(* PLC project batch, Dassault Systèmes ControlBuild 2024x Refresh1 *)
(* stored: creationDateTime 2024-03-18T16:40:20-01:00 *)

FUNCTION_BLOCK acknowledgepb
  VAR_IN_OUT
    action : BOOL := false;
    timeCounter : REAL := 0.0;
    pulseDuration : REAL := 0.0;
    PBLogic : BOOL := false;
  END_VAR
  VAR_OUTPUT
    PB : BOOL := false;
  END_VAR


ACTION C_source_code:

END_ACTION
END_FUNCTION_BLOCK

FUNCTION_BLOCK bpcloture
  VAR_IN_OUT
    action : BOOL := false;
    timeCounter : REAL := 0.0;
    pulseDuration : REAL := 0.0;
    PBLogic : BOOL := false;
  END_VAR
  VAR_OUTPUT
    PB : BOOL := false;
  END_VAR


ACTION C_source_code:

END_ACTION
END_FUNCTION_BLOCK

FUNCTION_BLOCK emergencystop
  VAR_IN_OUT
    action : BOOL := false;
    PBLogic : BOOL := false;
  END_VAR
  VAR_OUTPUT
    pb : BOOL := false;
  END_VAR


ACTION C_source_code:

END_ACTION
END_FUNCTION_BLOCK

FUNCTION_BLOCK endcyclepb
  VAR_IN_OUT
    action : BOOL := false;
    timeCounter : REAL := 0.0;
    pulseDuration : REAL := 0.0;
    PBLogic : BOOL := false;
  END_VAR
  VAR_OUTPUT
    PB : BOOL := false;
  END_VAR


ACTION C_source_code:

END_ACTION
END_FUNCTION_BLOCK

FUNCTION_BLOCK modeswitch
  VAR_IN_OUT
    leftPosition : BOOL := false;
    rightPosition : BOOL := false;
  END_VAR
  VAR_OUTPUT
    leftVariable : BOOL := false;
    rightVariable : BOOL := false;
  END_VAR


ACTION C_source_code:

END_ACTION
END_FUNCTION_BLOCK

FUNCTION_BLOCK powerup
  VAR_IN_OUT
    action : BOOL := false;
    timeCounter : REAL := 0.0;
    pulseDuration : REAL := 0.0;
    PBLogic : BOOL := false;
  END_VAR
  VAR_OUTPUT
    PB : BOOL := false;
  END_VAR


ACTION C_source_code:

END_ACTION
END_FUNCTION_BLOCK

FUNCTION_BLOCK startcyclepb
  VAR_IN_OUT
    action : BOOL := false;
    timeCounter : REAL := 0.0;
    pulseDuration : REAL := 0.0;
    PBLogic : BOOL := false;
  END_VAR
  VAR_OUTPUT
    PB : BOOL := false;
  END_VAR


ACTION C_source_code:

END_ACTION
END_FUNCTION_BLOCK

PROGRAM generalpanel
  VAR_OUTPUT
    acknowledgePB : BOOL := false;
    powerUp : BOOL := false;
    emergencyStop : BOOL := false;
    manualSwitch : BOOL := false;
    autoSwitch : BOOL := false;
    startCyclePB : BOOL := false;
    endCyclePB : BOOL := false;
  END_VAR

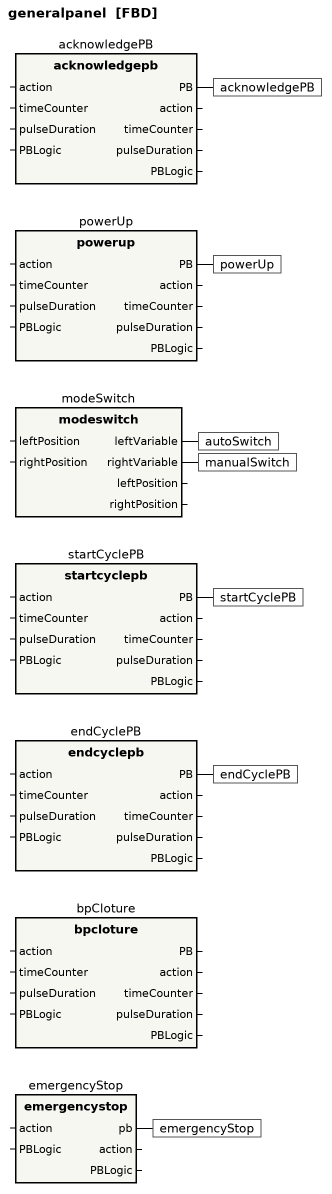
(* FBD diagram, written out as Structured Text *)
acknowledgePB();
acknowledgePB := acknowledgePB.PB;
powerUp();
powerUp := powerUp.PB;
emergencyStop();
emergencyStop := emergencyStop.pb;
modeSwitch();
manualSwitch := modeSwitch.rightVariable;
autoSwitch := modeSwitch.leftVariable;
startCyclePB();
startCyclePB := startCyclePB.PB;
endCyclePB();
endCyclePB := endCyclePB.PB;
bpCloture();
END_PROGRAM

FUNCTION_BLOCK management
  VAR_INPUT
    cycleInProgress : BOOL := false;
    endCycleRequest : BOOL := false;
    kneadingOk : BOOL := false;
    syrupWeighingOk : BOOL := false;
    flourWeighingOk : BOOL := false;
  END_VAR
  VAR_OUTPUT
    cycleEnd : BOOL := false;
    flourWeighingRq : BOOL := false;
    syrupWeighingRq : BOOL := false;
    kneadingRq : BOOL := false;
  END_VAR


ACTION C_source_code:

END_ACTION
END_FUNCTION_BLOCK

FUNCTION_BLOCK faults1
  VAR_INPUT
    closeCmd : BOOL := false;
    openCmd : BOOL := false;
    closedSensorFB : BOOL := false;
    openedSensorFB : BOOL := false;
    acknowledgePB : BOOL := false;
    thermalFB : Unknown := ();
    cmdFB : Unknown := ();
    cmd : Unknown := ();
    generalFault1 : Unknown := ();
    generalFault2 : Unknown := ();
    generalFault3 : Unknown := ();
    generalFault4 : Unknown := ();
  END_VAR
  VAR_IN_OUT
    closedSensorFault : BOOL := false;
    openedSensorFault : BOOL := false;
    discordanceFault : BOOL := false;
    ton_sec_1_i_ton : INT := 0;
    ton_sec_1_t1_ton : REAL := 0.0;
    ton_sec_1_t2_ton : INT := 0;
    ton_sec_1_Q : BOOL := false;
    ton_sec_1_CV : INT := 0;
    ton_sec_2_i_ton : INT := 0;
    ton_sec_2_t1_ton : REAL := 0.0;
    ton_sec_2_t2_ton : INT := 0;
    ton_sec_2_Q : BOOL := false;
    ton_sec_2_CV : INT := 0;
    ton_ms_3_i_tonms : INT := 0;
    ton_ms_3_t1_tonms : REAL := 0.0;
    ton_ms_3_t2_tonms : INT := 0;
    ton_ms_3_Q : BOOL := false;
    ton_ms_3_CV : INT := 0;
    presetMvt : ANY_STRING := ();
    presetDiscordance : ANY_STRING := ();
  END_VAR
  VAR_OUTPUT
    generalFault : BOOL := false;
    fault : BOOL := false;
  END_VAR


ACTION C_source_code:

END_ACTION
END_FUNCTION_BLOCK

FUNCTION_BLOCK actions
  VAR_INPUT
    autoMode : BOOL := false;
    manualMode : BOOL := false;
    autoCloseCmd : BOOL := false;
    autoOpenCmd : BOOL := false;
    closedSensorFB : BOOL := false;
    openedSensorFB : BOOL := false;
    closeValvePB : BOOL := false;
    openValvePB : BOOL := false;
    generalFault : BOOL := false;
    autoCmd : Unknown := ();
    forwardPB : Unknown := ();
    stopPB : Unknown := ();
  END_VAR
  VAR_OUTPUT
    closeCmd : BOOL := false;
    openCmd : BOOL := false;
    cmd : BOOL := false;
  END_VAR


ACTION C_source_code:

END_ACTION
END_FUNCTION_BLOCK

PROGRAM cmdofvalve
  VAR_INPUT
    autoMode : BOOL := false;
    manualMode : BOOL := false;
    closedSensorFB : BOOL := false;
    openedSensorFB : BOOL := false;
    autoCloseCmd : BOOL := false;
    autoOpenCmd : BOOL := false;
    closeValvePB : BOOL := false;
    openValvePB : BOOL := false;
    acknowledgePB : BOOL := false;
  END_VAR
  VAR_OUTPUT
    closeCmd : BOOL := false;
    openCmd : BOOL := false;
    generalFault : BOOL := false;
  END_VAR

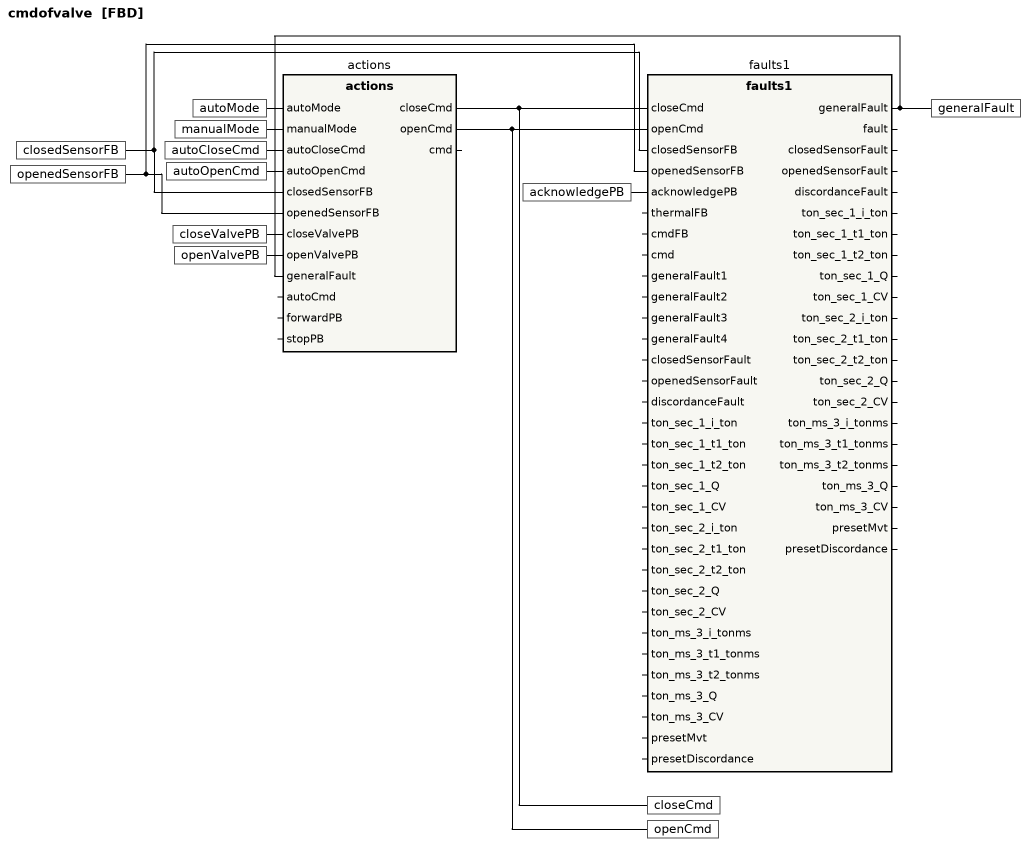
(* FBD diagram, written out as Structured Text *)
faults1(closeCmd := actions.closeCmd, openCmd := actions.openCmd, closedSensorFB := closedSensorFB, openedSensorFB := openedSensorFB, acknowledgePB := acknowledgePB);
actions(autoMode := autoMode, manualMode := manualMode, autoCloseCmd := autoCloseCmd, autoOpenCmd := autoOpenCmd, closedSensorFB := closedSensorFB, openedSensorFB := openedSensorFB, closeValvePB := closeValvePB, openValvePB := openValvePB, generalFault := faults1.generalFault);
closeCmd := actions.closeCmd;
openCmd := actions.openCmd;
generalFault := faults1.generalFault;
END_PROGRAM

FUNCTION_BLOCK switch
  VAR_IN_OUT
    leftPosition : BOOL := false;
    middlePosition : BOOL := false;
    rightPosition : BOOL := false;
  END_VAR
  VAR_OUTPUT
    leftVariable : BOOL := false;
    rightVariable : BOOL := false;
  END_VAR


ACTION C_source_code:

END_ACTION
END_FUNCTION_BLOCK

PROGRAM panel1
  VAR_OUTPUT
    closeValvePB : BOOL := false;
    openValvePB : BOOL := false;
    stopPB : BOOL := false;
    forwardPB : BOOL := false;
  END_VAR

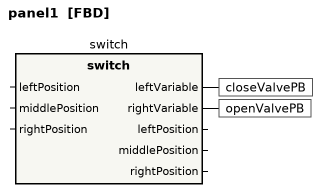
(* FBD diagram, written out as Structured Text *)
switch();
closeValvePB := switch.leftVariable;
openValvePB := switch.rightVariable;
END_PROGRAM

FUNCTION_BLOCK valve
  VAR_INPUT
    voltage380 : BOOL := false;
    cmdSupply : BOOL := false;
    sensorSupply : BOOL := false;
    openCmd : BOOL := false;
    closeCmd : BOOL := false;
    inputFlow : REAL := 0.0;
  END_VAR
  VAR_IN_OUT
    increment : REAL := 0.0;
    memoOpen : BOOL := false;
    memoClose : BOOL := false;
    openState : BOOL := false;
    closeState : BOOL := false;
    openingVal : REAL := 0.0;
    unit : REAL := 0.0;
    openingTime : REAL := 0.0;
    openedSensorLogic : BOOL := false;
    closedSensorLogic : BOOL := false;
    flowMax : REAL := 0.0;
    flowPerHour : BOOL := false;
    flowPerMinute : BOOL := false;
    d_locking : BOOL := false;
    v_d_locking : REAL := 0.0;
    d_flow : BOOL := false;
    v_d_flow : REAL := 0.0;
    d_electrical : BOOL := false;
    v_d_electrical : BOOL := false;
    d_closedSensor : BOOL := false;
    v_d_closedSensor : BOOL := false;
    d_openedSensor : BOOL := false;
    v_d_openedSensor : BOOL := false;
  END_VAR
  VAR_OUTPUT
    openedSensor : BOOL := false;
    closedSensor : BOOL := false;
    outputFlow : REAL := 0.0;
    percentOpening : REAL := 0.0;
  END_VAR


ACTION C_source_code:

END_ACTION
END_FUNCTION_BLOCK

PROGRAM airarrival
  VAR_INPUT
    acknowledgePB : BOOL := false;
    autoMode : BOOL := false;
    manualMode : BOOL := false;
    autoCloseCmd : BOOL := false;
    autoOpenCmd : BOOL := false;
    inputFlow : REAL := 0.0;
  END_VAR
  VAR_OUTPUT
    openedSensor : BOOL := false;
    closedSensor : BOOL := false;
    generalFault : BOOL := false;
    outputFlow : REAL := 0.0;
    percentOpening : REAL := 0.0;
  END_VAR

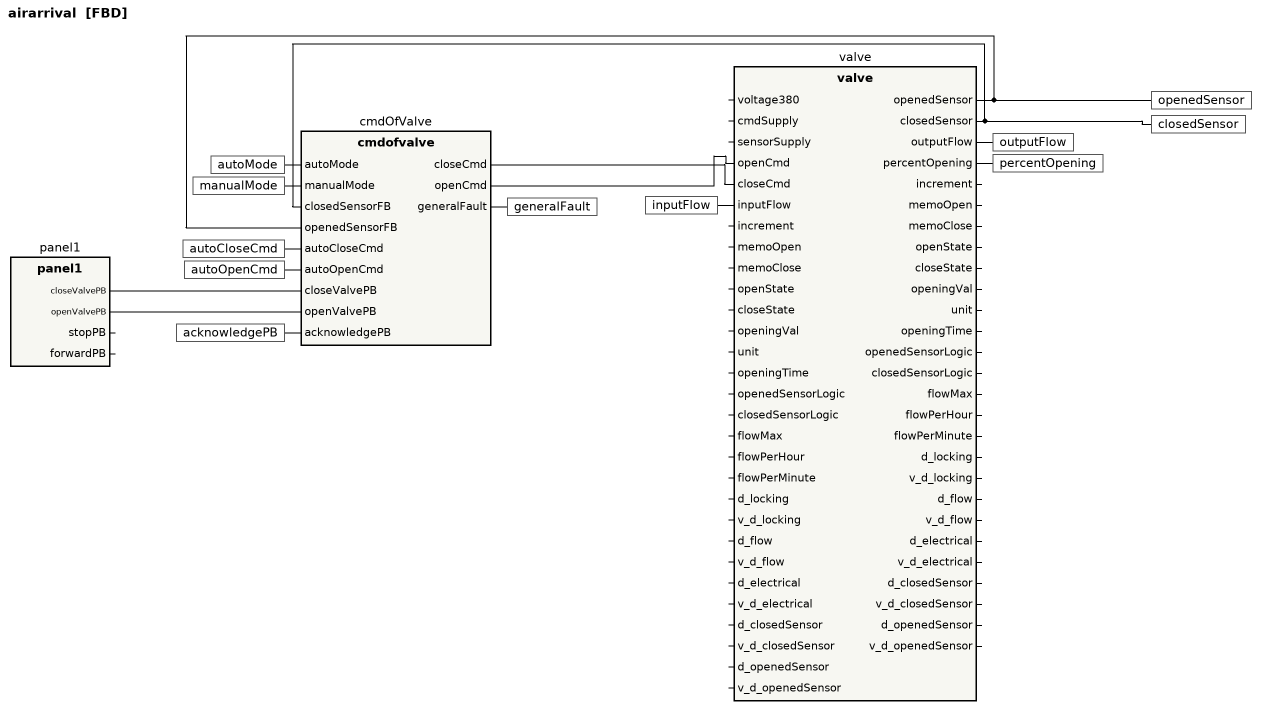
(* FBD diagram, written out as Structured Text *)
panel1();
cmdOfValve(autoMode := autoMode, manualMode := manualMode, closedSensorFB := valve.closedSensor, openedSensorFB := valve.openedSensor, autoCloseCmd := autoCloseCmd, autoOpenCmd := autoOpenCmd, closeValvePB := panel1.closeValvePB, openValvePB := panel1.openValvePB, acknowledgePB := acknowledgePB);
valve(openCmd := cmdOfValve.openCmd, closeCmd := cmdOfValve.closeCmd, inputFlow := inputFlow);
openedSensor := valve.openedSensor;
closedSensor := valve.closedSensor;
generalFault := cmdOfValve.generalFault;
outputFlow := valve.outputFlow;
percentOpening := valve.percentOpening;
END_PROGRAM

PROGRAM airextraction
  VAR_INPUT
    acknowledgePB : BOOL := false;
    autoMode : BOOL := false;
    manualMode : BOOL := false;
    autoCloseCmd : BOOL := false;
    autoOpenCmd : BOOL := false;
    inputFlow : REAL := 0.0;
  END_VAR
  VAR_OUTPUT
    openedSensor : BOOL := false;
    closedSensor : BOOL := false;
    generalFault : BOOL := false;
    outputFlow : REAL := 0.0;
    percentOpening : REAL := 0.0;
  END_VAR

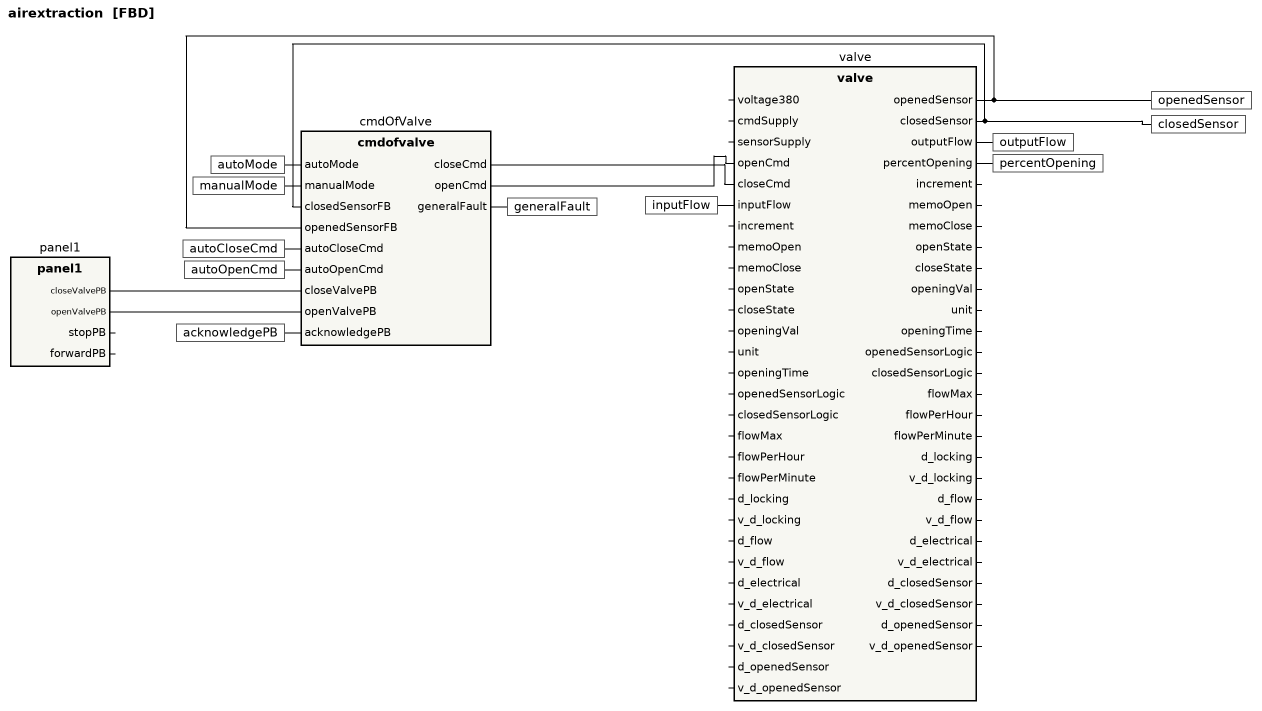
(* FBD diagram, written out as Structured Text *)
panel1();
cmdOfValve(autoMode := autoMode, manualMode := manualMode, closedSensorFB := valve.closedSensor, openedSensorFB := valve.openedSensor, autoCloseCmd := autoCloseCmd, autoOpenCmd := autoOpenCmd, closeValvePB := panel1.closeValvePB, openValvePB := panel1.openValvePB, acknowledgePB := acknowledgePB);
valve(openCmd := cmdOfValve.openCmd, closeCmd := cmdOfValve.closeCmd, inputFlow := inputFlow);
openedSensor := valve.openedSensor;
closedSensor := valve.closedSensor;
generalFault := cmdOfValve.generalFault;
outputFlow := valve.outputFlow;
percentOpening := valve.percentOpening;
END_PROGRAM

PROGRAM extractingvalve
  VAR_INPUT
    acknowledgePB : BOOL := false;
    autoMode : BOOL := false;
    manualMode : BOOL := false;
    autoCloseCmd : BOOL := false;
    autoOpenCmd : BOOL := false;
    inputFlow : REAL := 0.0;
  END_VAR
  VAR_OUTPUT
    openedSensor : BOOL := false;
    closedSensor : BOOL := false;
    generalFault : BOOL := false;
    outputFlow : REAL := 0.0;
    percentOpening : REAL := 0.0;
  END_VAR

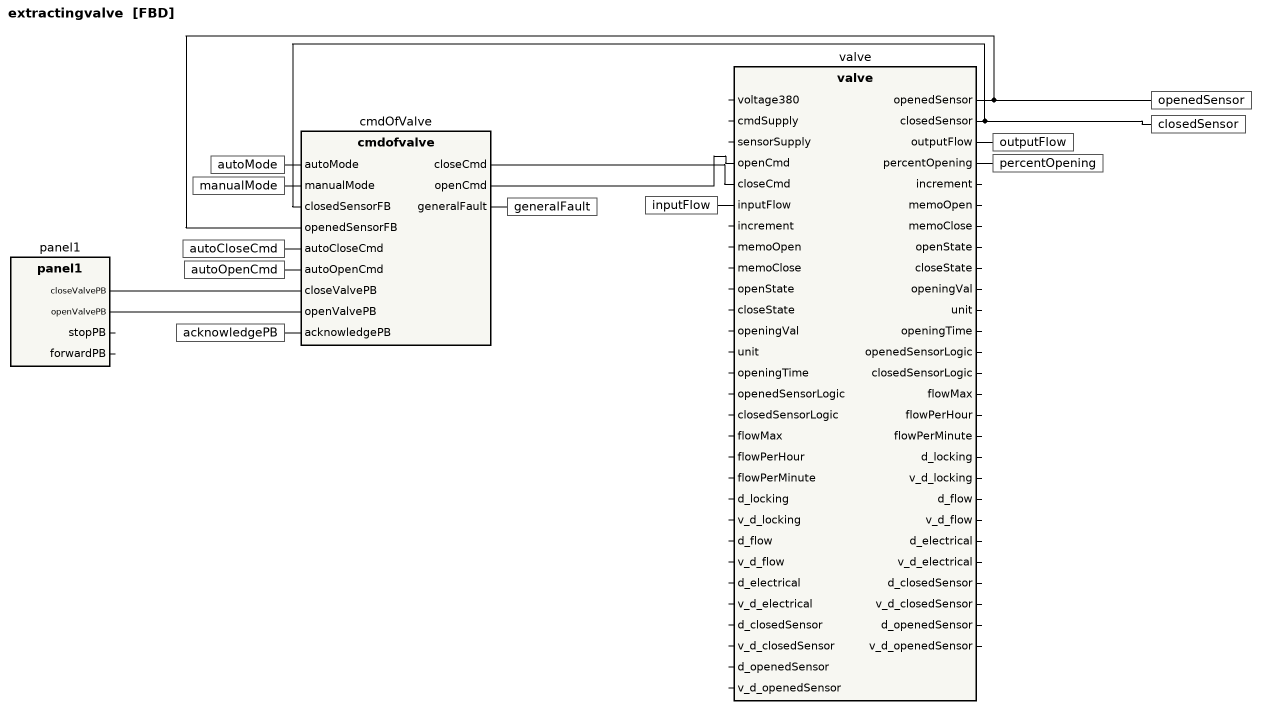
(* FBD diagram, written out as Structured Text *)
panel1();
cmdOfValve(autoMode := autoMode, manualMode := manualMode, closedSensorFB := valve.closedSensor, openedSensorFB := valve.openedSensor, autoCloseCmd := autoCloseCmd, autoOpenCmd := autoOpenCmd, closeValvePB := panel1.closeValvePB, openValvePB := panel1.openValvePB, acknowledgePB := acknowledgePB);
valve(openCmd := cmdOfValve.openCmd, closeCmd := cmdOfValve.closeCmd, inputFlow := inputFlow);
openedSensor := valve.openedSensor;
closedSensor := valve.closedSensor;
generalFault := cmdOfValve.generalFault;
outputFlow := valve.outputFlow;
percentOpening := valve.percentOpening;
END_PROGRAM

FUNCTION_BLOCK flourmanagement
  VAR_INPUT
    weighingRequest : BOOL := false;
    cycleInProgress : BOOL := false;
    weighedWeight : INT := 0;
    flourWeight : INT := 0;
  END_VAR
  VAR_IN_OUT
    totalWeight : INT := 0;
    endOfWeighing : BOOL := false;
    maxWeight : INT := 0;
  END_VAR
  VAR_OUTPUT
    weighingOk : BOOL := false;
    introduceFlour : BOOL := false;
    introFlourEnd : BOOL := false;
    exitFlour : BOOL := false;
    exitFlourEnd : BOOL := false;
  END_VAR


ACTION C_source_code:

END_ACTION
END_FUNCTION_BLOCK

FUNCTION_BLOCK flourweighing
  VAR_INPUT
    inletFlow : REAL := 0.0;
    outletFlow : REAL := 0.0;
  END_VAR
  VAR_IN_OUT
    percent : REAL := 0.0;
    capacity : REAL := 0.0;
    d_level : BOOL := false;
    v_d_level : REAL := 0.0;
  END_VAR
  VAR_OUTPUT
    tankLevel : REAL := 0.0;
  END_VAR


ACTION C_source_code:

END_ACTION
END_FUNCTION_BLOCK

FUNCTION_BLOCK flow
  VAR_INPUT
    inputFlow : REAL := 0.0;
  END_VAR
  VAR_IN_OUT
    unit : REAL := 0.0;
    flowMax : REAL := 0.0;
    flowPerHour : BOOL := false;
    flowPerMinute : BOOL := false;
  END_VAR
  VAR_OUTPUT
    outputFlow : REAL := 0.0;
  END_VAR


ACTION C_source_code:

END_ACTION
END_FUNCTION_BLOCK

FUNCTION_BLOCK level
  VAR_INPUT
    measure : REAL := 0.0;
    sensorSupply : BOOL := false;
  END_VAR
  VAR_IN_OUT
    tmp : INT := 0;
    localValue : REAL := 0.0;
    nbDigit : BOOL := false;
    d_value : BOOL := false;
    v_d_value : REAL := 0.0;
  END_VAR
  VAR_OUTPUT
    realValue : REAL := 0.0;
    intValue : REAL := 0.0;
    dintValue : REAL := 0.0;
  END_VAR


ACTION C_source_code:

END_ACTION
END_FUNCTION_BLOCK

FUNCTION_BLOCK scale
  VAR_INPUT
    inputValue : REAL := 0.0;
  END_VAR
  VAR_IN_OUT
    a : REAL := 0.0;
    b : REAL := 0.0;
    k : REAL := 0.0;
    minInput : REAL := 0.0;
    maxInput : REAL := 0.0;
    minOutput : REAL := 0.0;
    maxOutput : REAL := 0.0;
    d_scale : BOOL := false;
    v_d_scale : REAL := 0.0;
  END_VAR
  VAR_OUTPUT
    realValue : REAL := 0.0;
    dintValue : INT := 0;
    intValue : INT := 0;
  END_VAR


ACTION C_source_code:

END_ACTION
END_FUNCTION_BLOCK

PROGRAM flour
  VAR_INPUT
    cycleInProgress : BOOL := false;
    acknowledgePB : BOOL := false;
    weighingRequest : BOOL := false;
    flourWeight : INT := 0;
    autoMode : BOOL := false;
    manualMode : BOOL := false;
  END_VAR
  VAR_OUTPUT
    flourExtraction : REAL := 0.0;
    weighingOk : BOOL := false;
    fault : BOOL := false;
  END_VAR

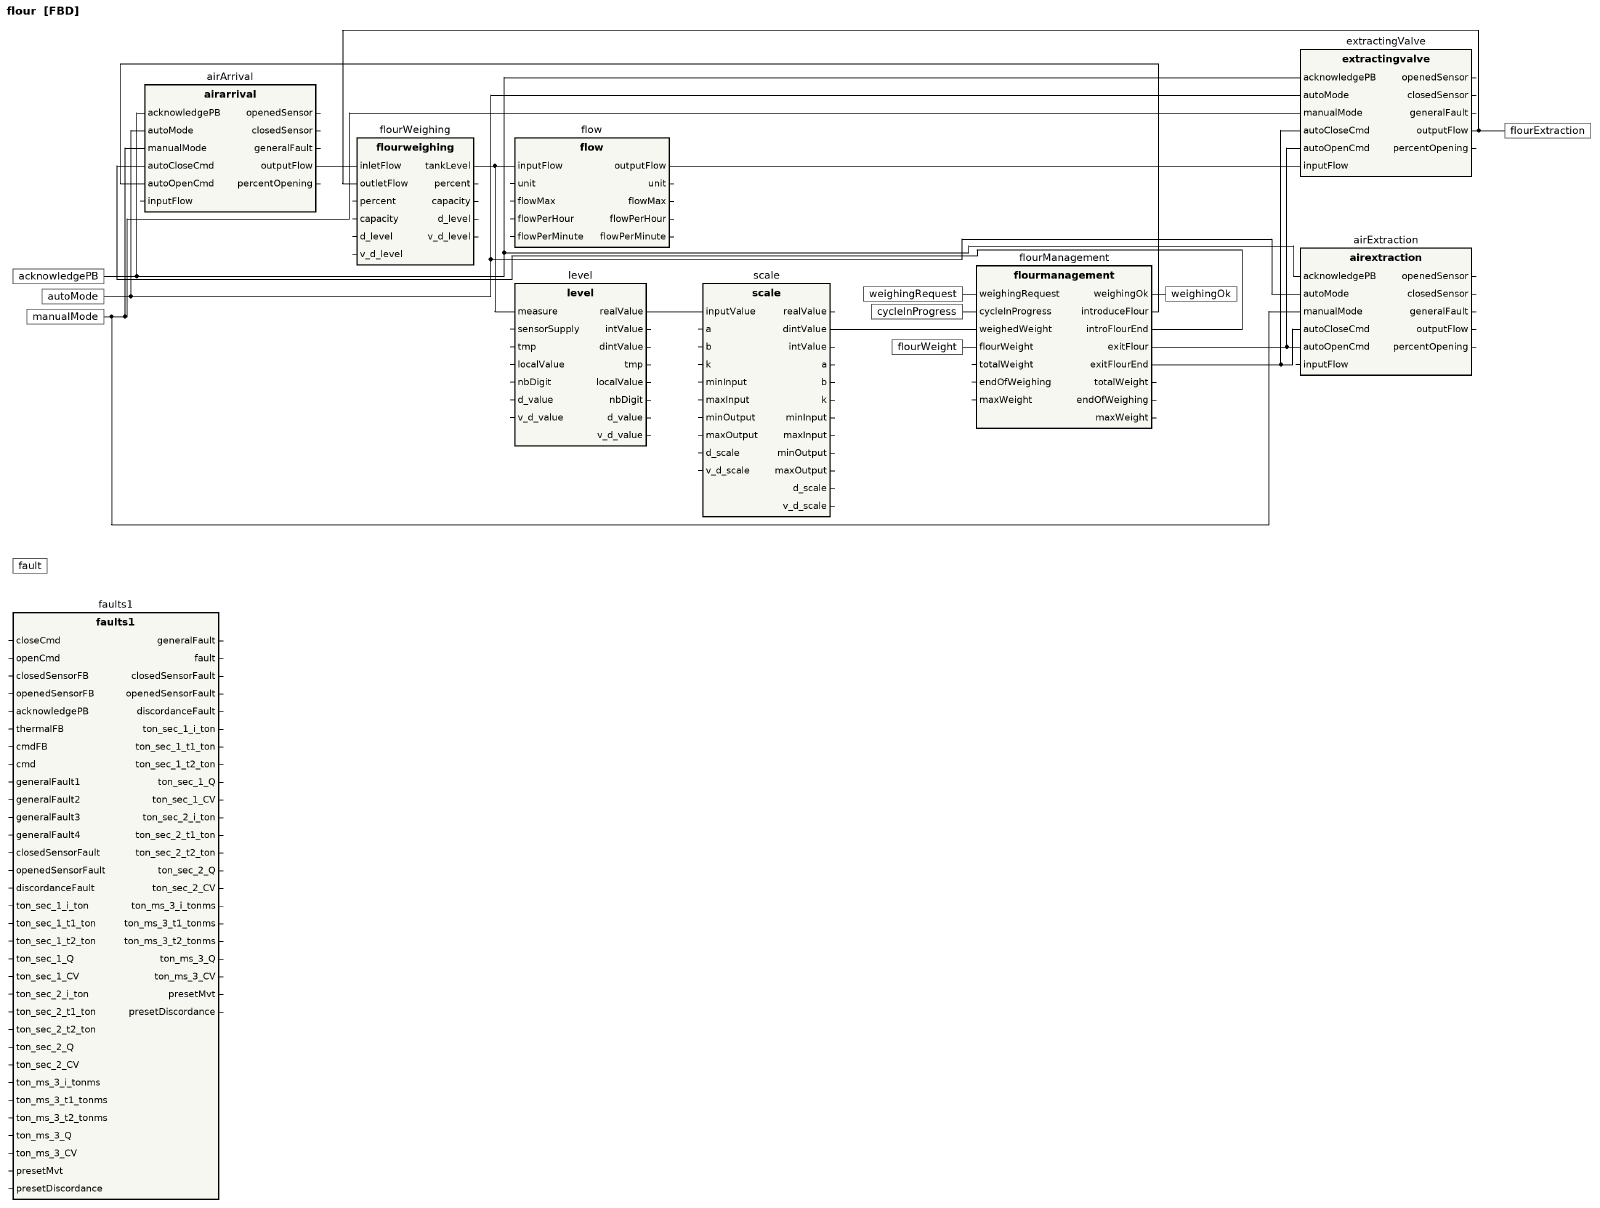
(* FBD diagram, written out as Structured Text *)
airArrival(acknowledgePB := acknowledgePB, autoMode := autoMode, manualMode := manualMode, autoCloseCmd := flourManagement.introFlourEnd, autoOpenCmd := flourManagement.introduceFlour);
flourWeighing(inletFlow := airArrival.outputFlow, outletFlow := extractingValve.outputFlow);
level(measure := flourWeighing.tankLevel);
scale(inputValue := level.realValue);
flourManagement(weighingRequest := weighingRequest, cycleInProgress := cycleInProgress, weighedWeight := scale.dintValue, flourWeight := flourWeight);
flow(inputFlow := flourWeighing.tankLevel);
extractingValve(acknowledgePB := acknowledgePB, autoMode := autoMode, manualMode := manualMode, autoCloseCmd := flourManagement.exitFlourEnd, autoOpenCmd := flourManagement.exitFlour, inputFlow := flow.outputFlow);
flourExtraction := extractingValve.outputFlow;
weighingOk := flourManagement.weighingOk;
airExtraction(acknowledgePB := acknowledgePB, autoMode := autoMode, manualMode := manualMode, autoCloseCmd := flourManagement.exitFlourEnd, autoOpenCmd := flourManagement.exitFlour);
faults1();
END_PROGRAM

PROGRAM cleaningvalve
  VAR_INPUT
    acknowledgePB : BOOL := false;
    autoMode : BOOL := false;
    manualMode : BOOL := false;
    autoCloseCmd : BOOL := false;
    autoOpenCmd : BOOL := false;
    inputFlow : REAL := 0.0;
  END_VAR
  VAR_OUTPUT
    openedSensor : BOOL := false;
    closedSensor : BOOL := false;
    generalFault : BOOL := false;
    outputFlow : REAL := 0.0;
    percentOpening : REAL := 0.0;
  END_VAR

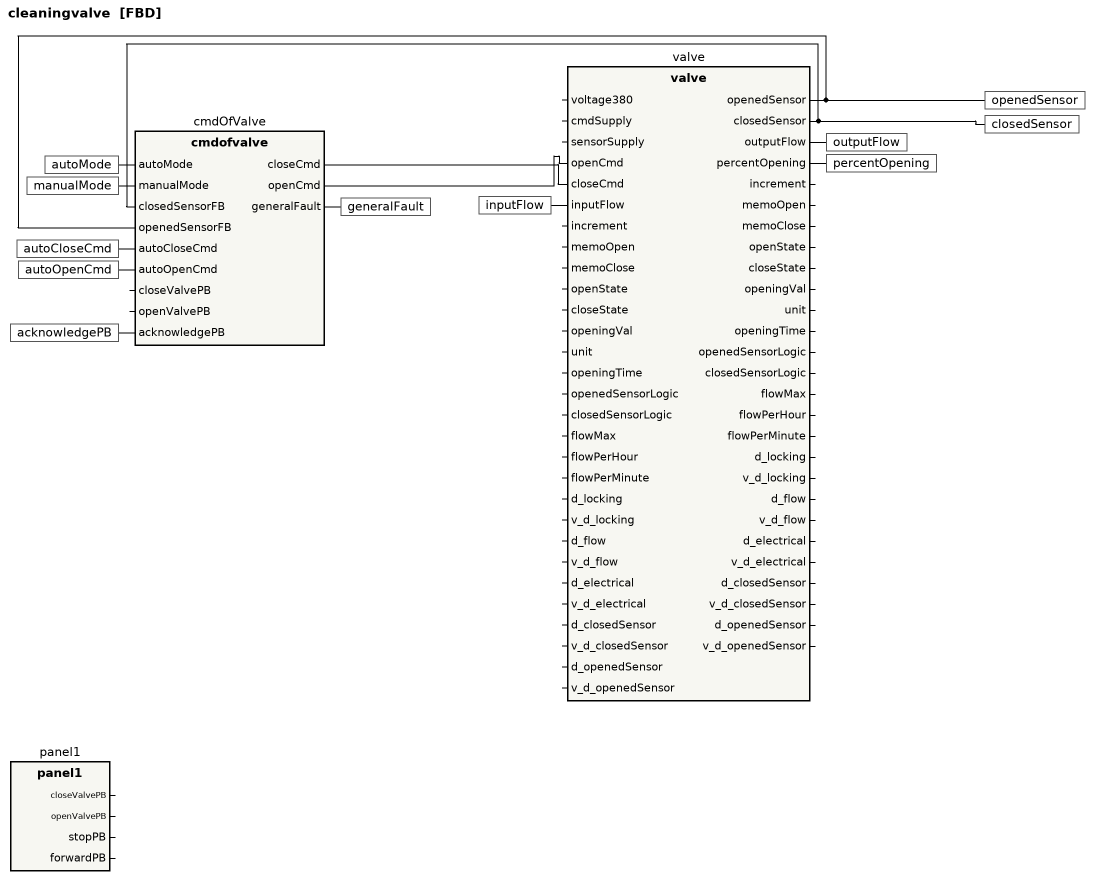
(* FBD diagram, written out as Structured Text *)
cmdOfValve(autoMode := autoMode, manualMode := manualMode, closedSensorFB := valve.closedSensor, openedSensorFB := valve.openedSensor, autoCloseCmd := autoCloseCmd, autoOpenCmd := autoOpenCmd, acknowledgePB := acknowledgePB);
valve(openCmd := cmdOfValve.openCmd, closeCmd := cmdOfValve.closeCmd, inputFlow := inputFlow);
openedSensor := valve.openedSensor;
closedSensor := valve.closedSensor;
generalFault := cmdOfValve.generalFault;
outputFlow := valve.outputFlow;
percentOpening := valve.percentOpening;
panel1();
END_PROGRAM

FUNCTION_BLOCK collectedmixture
  VAR_INPUT
    flowSyrup1 : REAL := 0.0;
    flowSyrup2 : REAL := 0.0;
    flowSyrup3 : REAL := 0.0;
  END_VAR
  VAR_OUTPUT
    flow : REAL := 0.0;
  END_VAR


ACTION C_source_code:

END_ACTION
END_FUNCTION_BLOCK

FUNCTION_BLOCK kneading
  VAR_INPUT
    kneadingRequest : BOOL := false;
    cycleInProgress : BOOL := false;
    mixtureLevel : INT := 0;
  END_VAR
  VAR_IN_OUT
    nbCycles : INT := 0;
    kneadingDuration : INT := 0;
    nbOfCleanCycles : INT := 0;
    cleaningDuration : INT := 0;
  END_VAR
  VAR_OUTPUT
    kneadingOK : BOOL := false;
    knead : BOOL := false;
    clean : BOOL := false;
    cleaningEnd : BOOL := false;
    evacuateMixture : BOOL := false;
    evacMixtureEnd : BOOL := false;
  END_VAR


ACTION C_source_code:

END_ACTION
END_FUNCTION_BLOCK

PROGRAM mixtureextractingvalve
  VAR_INPUT
    acknowledgePB : BOOL := false;
    autoMode : BOOL := false;
    manualMode : BOOL := false;
    autoCloseCmd : BOOL := false;
    autoOpenCmd : BOOL := false;
    inputFlow : REAL := 0.0;
  END_VAR
  VAR_OUTPUT
    openedSensor : BOOL := false;
    closedSensor : BOOL := false;
    generalFault : BOOL := false;
    outputFlow : REAL := 0.0;
    percentOpening : REAL := 0.0;
  END_VAR

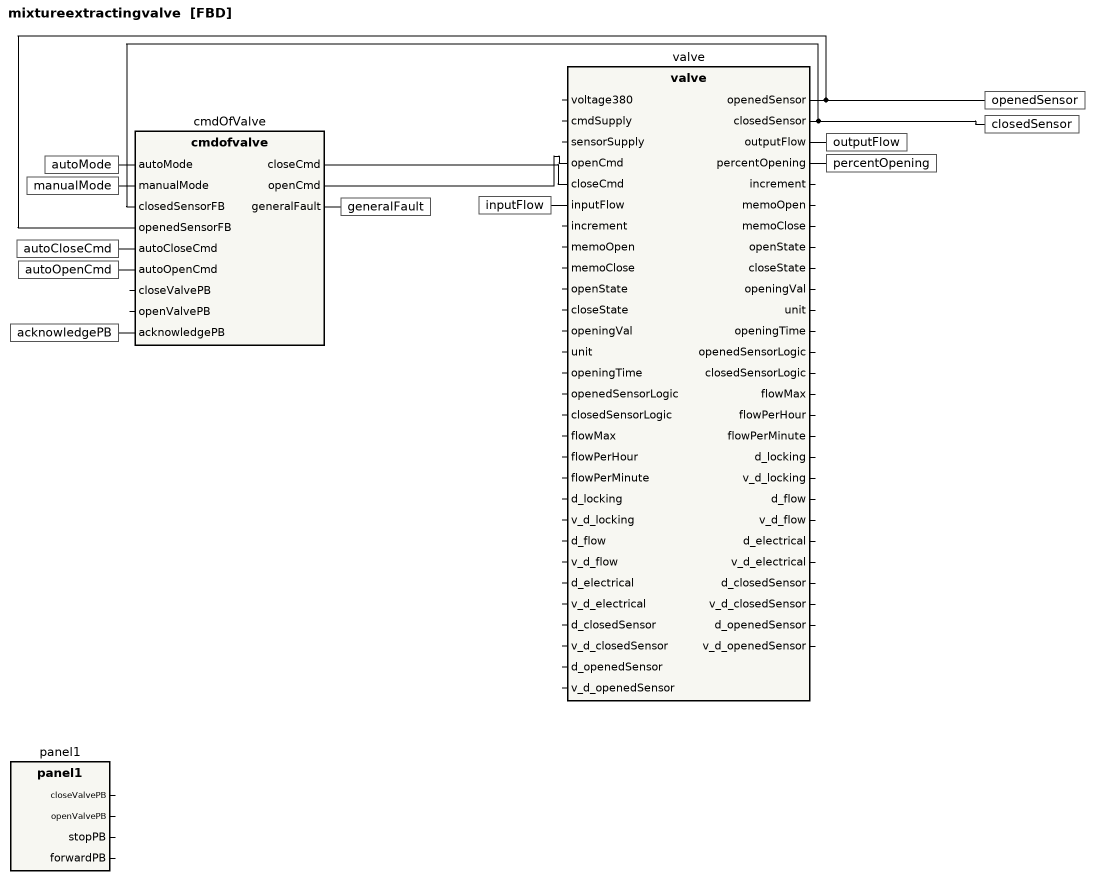
(* FBD diagram, written out as Structured Text *)
cmdOfValve(autoMode := autoMode, manualMode := manualMode, closedSensorFB := valve.closedSensor, openedSensorFB := valve.openedSensor, autoCloseCmd := autoCloseCmd, autoOpenCmd := autoOpenCmd, acknowledgePB := acknowledgePB);
valve(openCmd := cmdOfValve.openCmd, closeCmd := cmdOfValve.closeCmd, inputFlow := inputFlow);
openedSensor := valve.openedSensor;
closedSensor := valve.closedSensor;
generalFault := cmdOfValve.generalFault;
outputFlow := valve.outputFlow;
percentOpening := valve.percentOpening;
panel1();
END_PROGRAM

FUNCTION_BLOCK mixtureweighing
  VAR_INPUT
    inletFlow : REAL := 0.0;
    outletFlow : REAL := 0.0;
  END_VAR
  VAR_IN_OUT
    percent : REAL := 0.0;
    capacity : REAL := 0.0;
    d_level : BOOL := false;
    v_d_level : REAL := 0.0;
  END_VAR
  VAR_OUTPUT
    tankLevel : REAL := 0.0;
  END_VAR


ACTION C_source_code:

END_ACTION
END_FUNCTION_BLOCK

FUNCTION_BLOCK agitator
  VAR_INPUT
    voltage380 : BOOL := false;
    cmdSupply : BOOL := false;
    sensorSupply : BOOL := false;
    cmd : BOOL := false;
  END_VAR
  VAR_IN_OUT
    increment : REAL := 0.0;
    memo : BOOL := false;
    state : BOOL := false;
    speedSetpoint : REAL := 0.0;
    cnt : INT := 0;
    flipflop : BOOL := false;
    nominalTime : REAL := 0.0;
    thermalLogic : BOOL := false;
    cmdFbLogic : BOOL := false;
    nominalSpeed : REAL := 0.0;
    d_locking : BOOL := false;
    v_d_locking : REAL := 0.0;
    d_electrical : BOOL := false;
    v_d_electrical : BOOL := false;
    d_cmdFB : BOOL := false;
    v_d_cmdFB : BOOL := false;
  END_VAR
  VAR_OUTPUT
    cmdFB : BOOL := false;
    thermal : BOOL := false;
    speedVal : REAL := 0.0;
    speedPercent : REAL := 0.0;
  END_VAR


ACTION C_source_code:

END_ACTION
END_FUNCTION_BLOCK

PROGRAM cmdofmotor
  VAR_INPUT
    autoMode : BOOL := false;
    manualMode : BOOL := false;
    autoCmd : BOOL := false;
    thermalFB : BOOL := false;
    cmdFB : BOOL := false;
    forwardPB : BOOL := false;
    stopPB : BOOL := false;
    acknowledgePB : BOOL := false;
  END_VAR
  VAR_OUTPUT
    cmd : BOOL := false;
    generalFault : BOOL := false;
  END_VAR

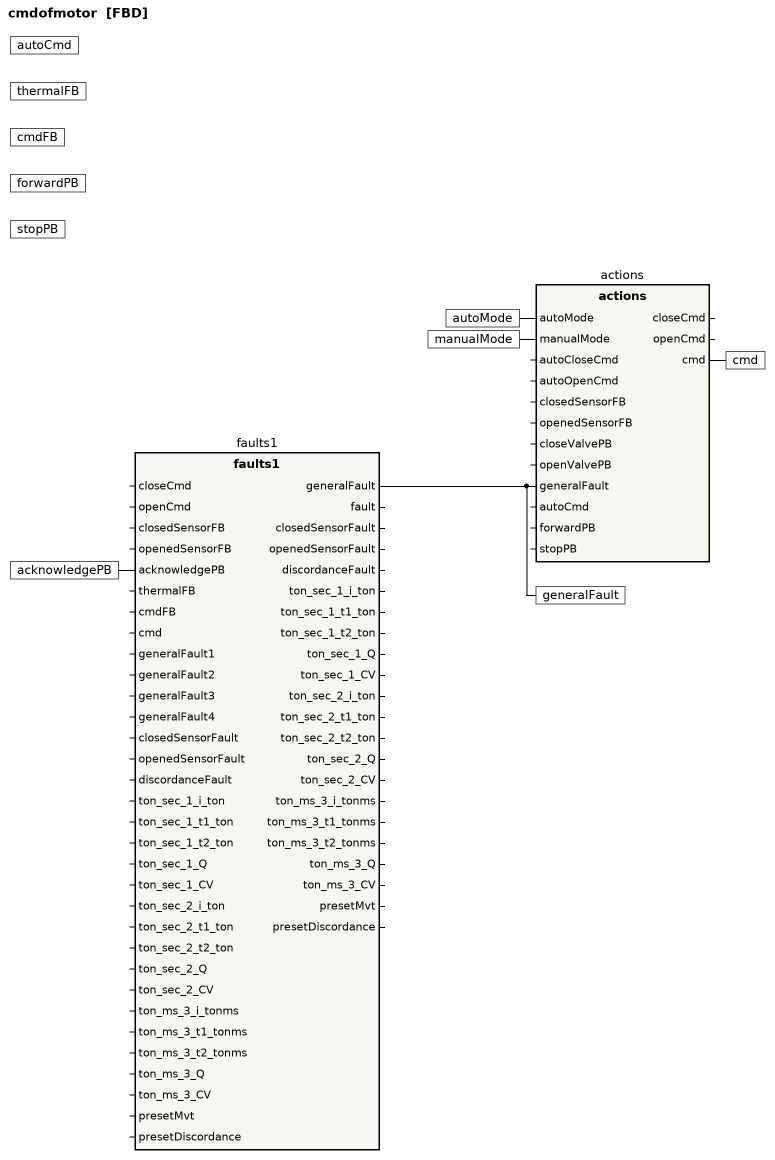
(* FBD diagram, written out as Structured Text *)
faults1(acknowledgePB := acknowledgePB);
actions(autoMode := autoMode, manualMode := manualMode, generalFault := faults1.generalFault);
cmd := actions.cmd;
generalFault := faults1.generalFault;
(* drawn but not wired to any output: autoCmd, thermalFB, cmdFB, forwardPB, stopPB *)
END_PROGRAM

PROGRAM motorofagitator
  VAR_INPUT
    acknowledgePB : BOOL := false;
    autoMode : BOOL := false;
    manualMode : BOOL := false;
    autoCmd : BOOL := false;
  END_VAR
  VAR_OUTPUT
    generalFault : BOOL := false;
    speedVal : REAL := 0.0;
    speedPercent : REAL := 0.0;
  END_VAR

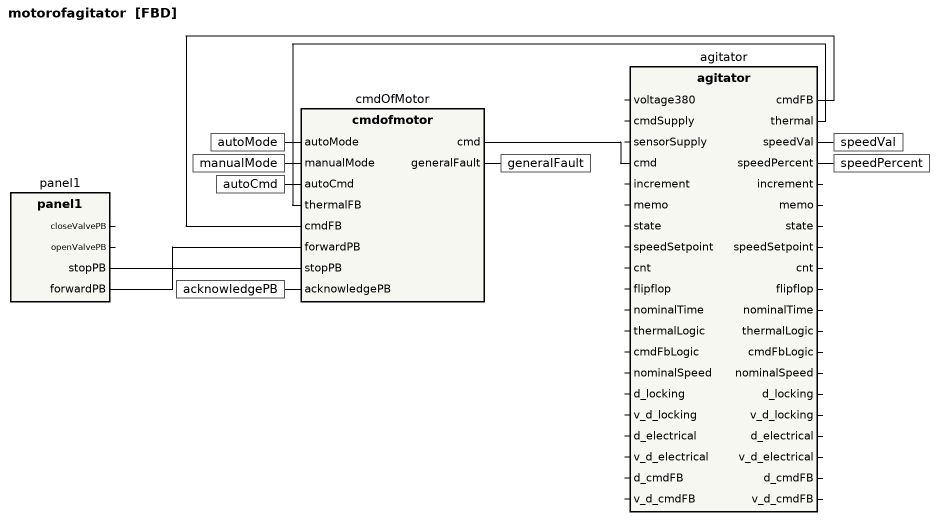
(* FBD diagram, written out as Structured Text *)
agitator(cmd := cmdOfMotor.cmd);
panel1();
cmdOfMotor(autoMode := autoMode, manualMode := manualMode, autoCmd := autoCmd, thermalFB := agitator.thermal, cmdFB := agitator.cmdFB, forwardPB := panel1.forwardPB, stopPB := panel1.stopPB, acknowledgePB := acknowledgePB);
generalFault := cmdOfMotor.generalFault;
speedVal := agitator.speedVal;
speedPercent := agitator.speedPercent;
END_PROGRAM

PROGRAM mixture
  VAR_INPUT
    cycleInProgress : BOOL := false;
    kneadingRequest : BOOL := false;
    acknowledgePB : BOOL := false;
    autoMode : BOOL := false;
    manualMode : BOOL := false;
    syrupExtraction : REAL := 0.0;
    flourExtraction : REAL := 0.0;
  END_VAR
  VAR_OUTPUT
    kneadingOK : BOOL := false;
    fault : BOOL := false;
  END_VAR

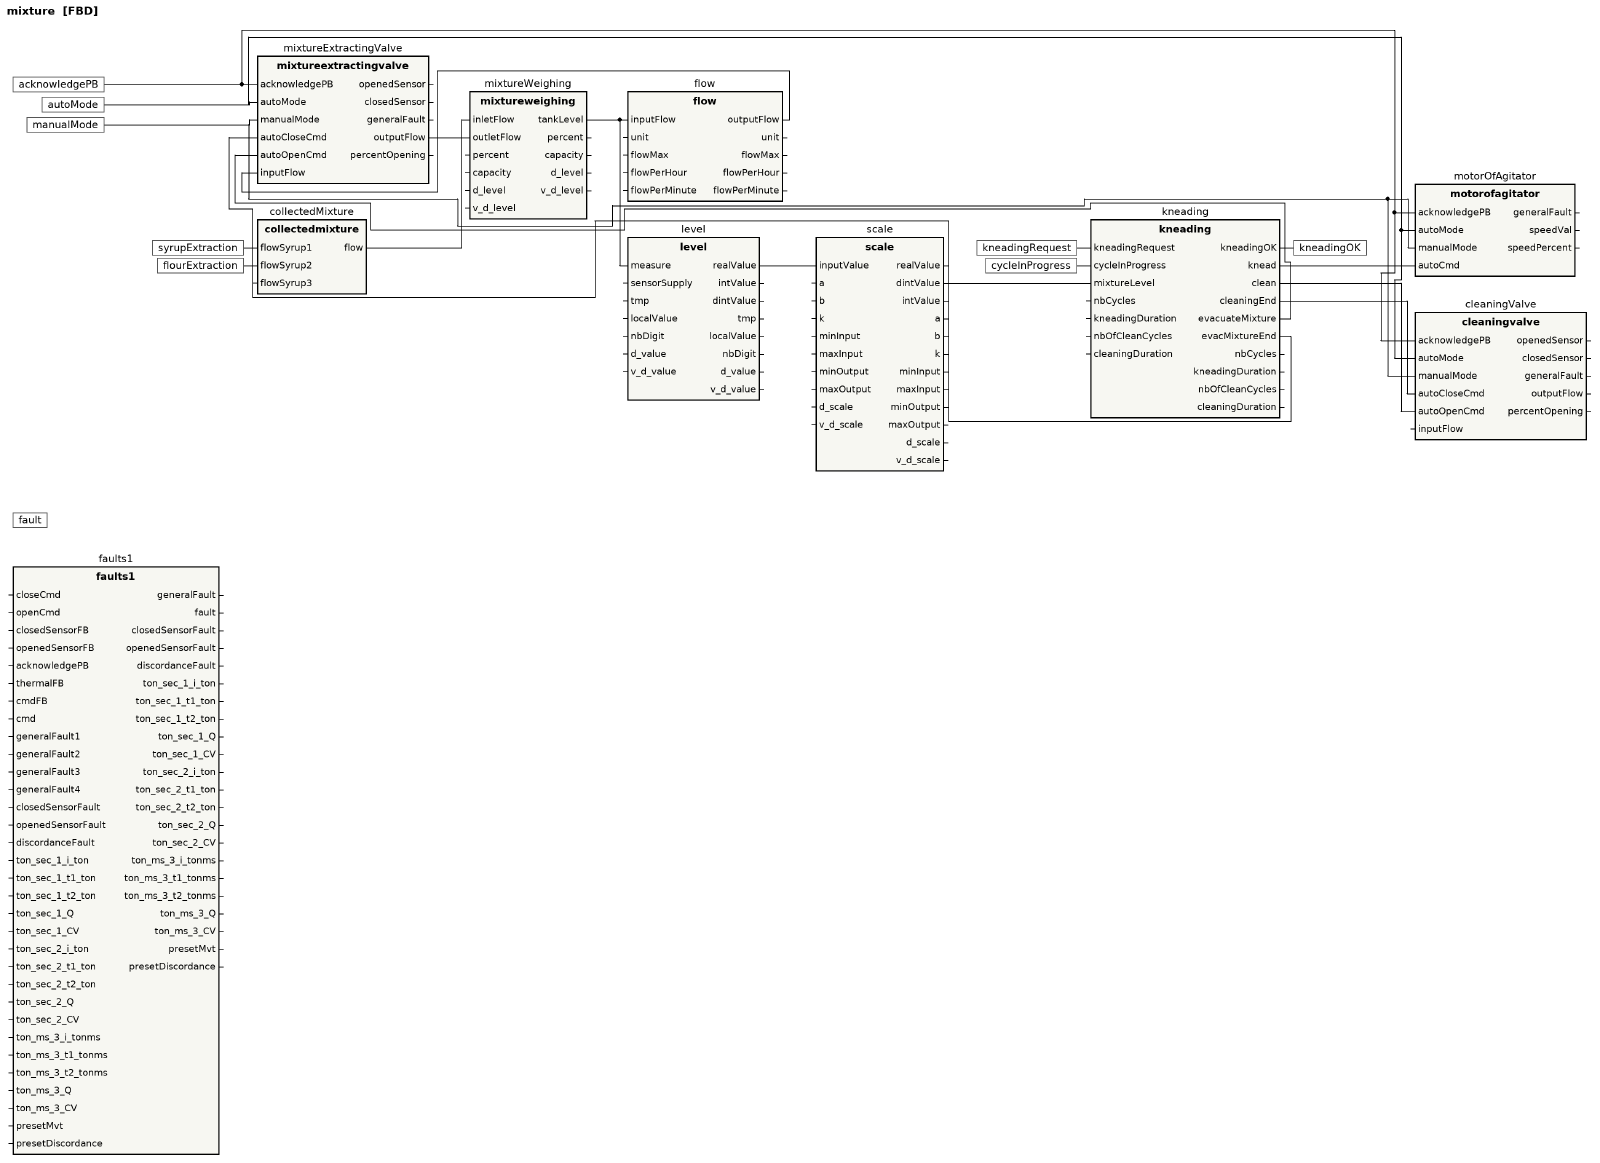
(* FBD diagram, written out as Structured Text *)
collectedMixture(flowSyrup1 := syrupExtraction, flowSyrup2 := flourExtraction);
flow(inputFlow := mixtureWeighing.tankLevel);
mixtureExtractingValve(acknowledgePB := acknowledgePB, autoMode := autoMode, manualMode := manualMode, autoCloseCmd := kneading.evacMixtureEnd, autoOpenCmd := kneading.evacuateMixture, inputFlow := flow.outputFlow);
mixtureWeighing(inletFlow := collectedMixture.flow, outletFlow := mixtureExtractingValve.outputFlow);
level(measure := mixtureWeighing.tankLevel);
scale(inputValue := level.realValue);
kneading(kneadingRequest := kneadingRequest, cycleInProgress := cycleInProgress, mixtureLevel := scale.dintValue);
kneadingOK := kneading.kneadingOK;
motorOfAgitator(acknowledgePB := acknowledgePB, autoMode := autoMode, manualMode := manualMode, autoCmd := kneading.knead);
faults1();
cleaningValve(acknowledgePB := acknowledgePB, autoMode := autoMode, manualMode := manualMode, autoCloseCmd := kneading.cleaningEnd, autoOpenCmd := kneading.clean);
END_PROGRAM

PROGRAM arrivalvalvesyrup1
  VAR_INPUT
    acknowledgePB : BOOL := false;
    autoMode : BOOL := false;
    manualMode : BOOL := false;
    autoCloseCmd : BOOL := false;
    autoOpenCmd : BOOL := false;
    inputFlow : REAL := 0.0;
  END_VAR
  VAR_OUTPUT
    openedSensor : BOOL := false;
    closedSensor : BOOL := false;
    generalFault : BOOL := false;
    outputFlow : REAL := 0.0;
    percentOpening : REAL := 0.0;
  END_VAR

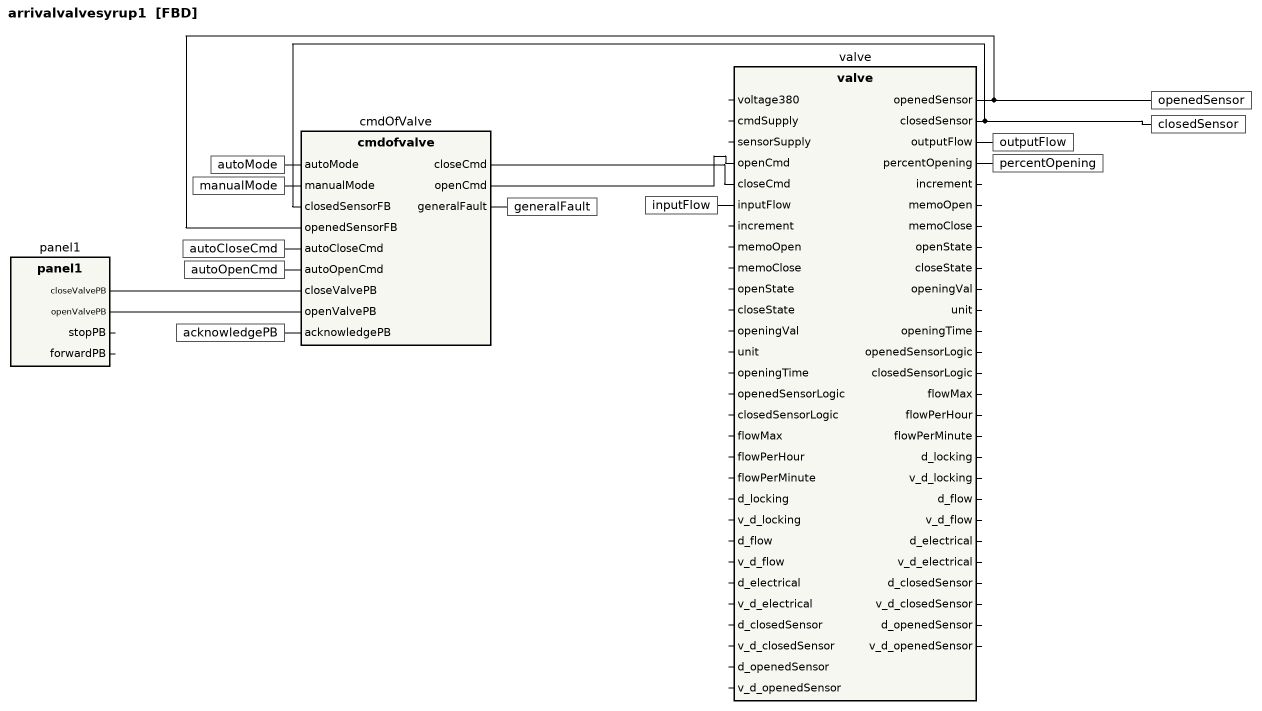
(* FBD diagram, written out as Structured Text *)
panel1();
cmdOfValve(autoMode := autoMode, manualMode := manualMode, closedSensorFB := valve.closedSensor, openedSensorFB := valve.openedSensor, autoCloseCmd := autoCloseCmd, autoOpenCmd := autoOpenCmd, closeValvePB := panel1.closeValvePB, openValvePB := panel1.openValvePB, acknowledgePB := acknowledgePB);
valve(openCmd := cmdOfValve.openCmd, closeCmd := cmdOfValve.closeCmd, inputFlow := inputFlow);
openedSensor := valve.openedSensor;
closedSensor := valve.closedSensor;
generalFault := cmdOfValve.generalFault;
outputFlow := valve.outputFlow;
percentOpening := valve.percentOpening;
END_PROGRAM

PROGRAM arrivalvalvesyrup2
  VAR_INPUT
    acknowledgePB : BOOL := false;
    autoMode : BOOL := false;
    manualMode : BOOL := false;
    autoCloseCmd : BOOL := false;
    autoOpenCmd : BOOL := false;
    inputFlow : REAL := 0.0;
  END_VAR
  VAR_OUTPUT
    openedSensor : BOOL := false;
    closedSensor : BOOL := false;
    generalFault : BOOL := false;
    outputFlow : REAL := 0.0;
    percentOpening : REAL := 0.0;
  END_VAR

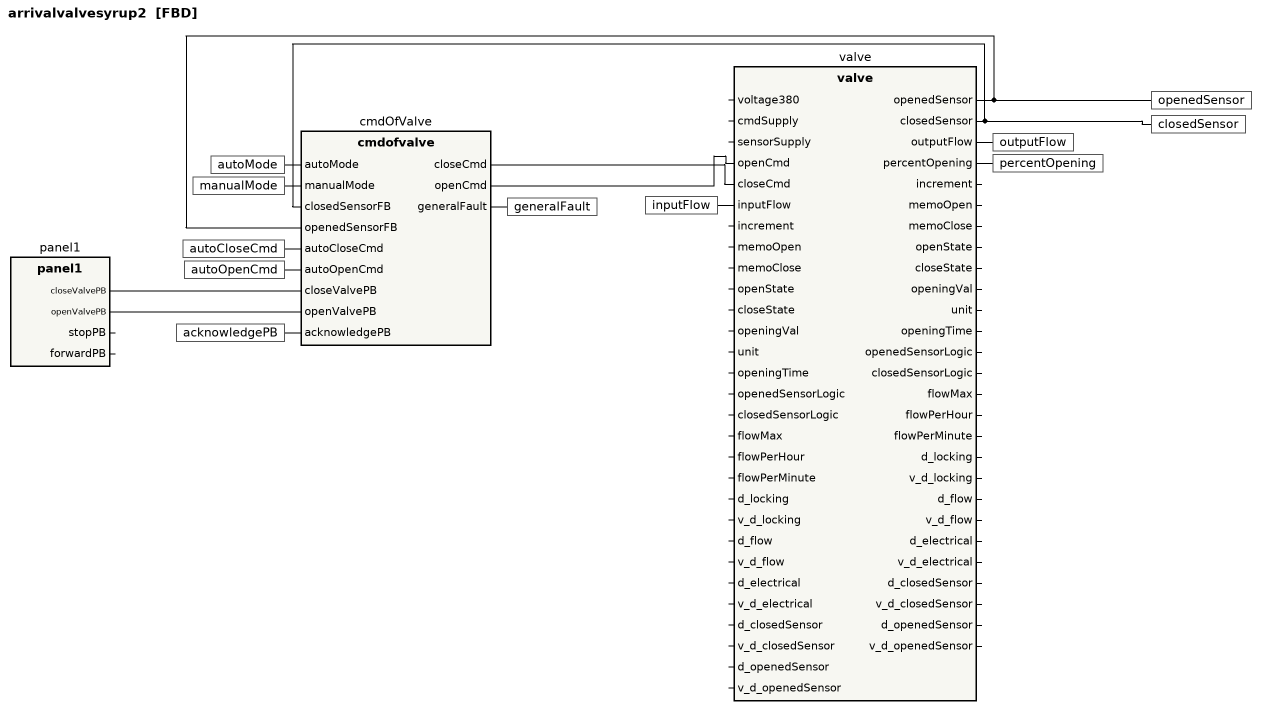
(* FBD diagram, written out as Structured Text *)
panel1();
cmdOfValve(autoMode := autoMode, manualMode := manualMode, closedSensorFB := valve.closedSensor, openedSensorFB := valve.openedSensor, autoCloseCmd := autoCloseCmd, autoOpenCmd := autoOpenCmd, closeValvePB := panel1.closeValvePB, openValvePB := panel1.openValvePB, acknowledgePB := acknowledgePB);
valve(openCmd := cmdOfValve.openCmd, closeCmd := cmdOfValve.closeCmd, inputFlow := inputFlow);
openedSensor := valve.openedSensor;
closedSensor := valve.closedSensor;
generalFault := cmdOfValve.generalFault;
outputFlow := valve.outputFlow;
percentOpening := valve.percentOpening;
END_PROGRAM

PROGRAM arrivalvalvesyrup3
  VAR_INPUT
    acknowledgePB : BOOL := false;
    autoMode : BOOL := false;
    manualMode : BOOL := false;
    autoCloseCmd : BOOL := false;
    autoOpenCmd : BOOL := false;
    inputFlow : REAL := 0.0;
  END_VAR
  VAR_OUTPUT
    openedSensor : BOOL := false;
    closedSensor : BOOL := false;
    generalFault : BOOL := false;
    outputFlow : REAL := 0.0;
    percentOpening : REAL := 0.0;
  END_VAR

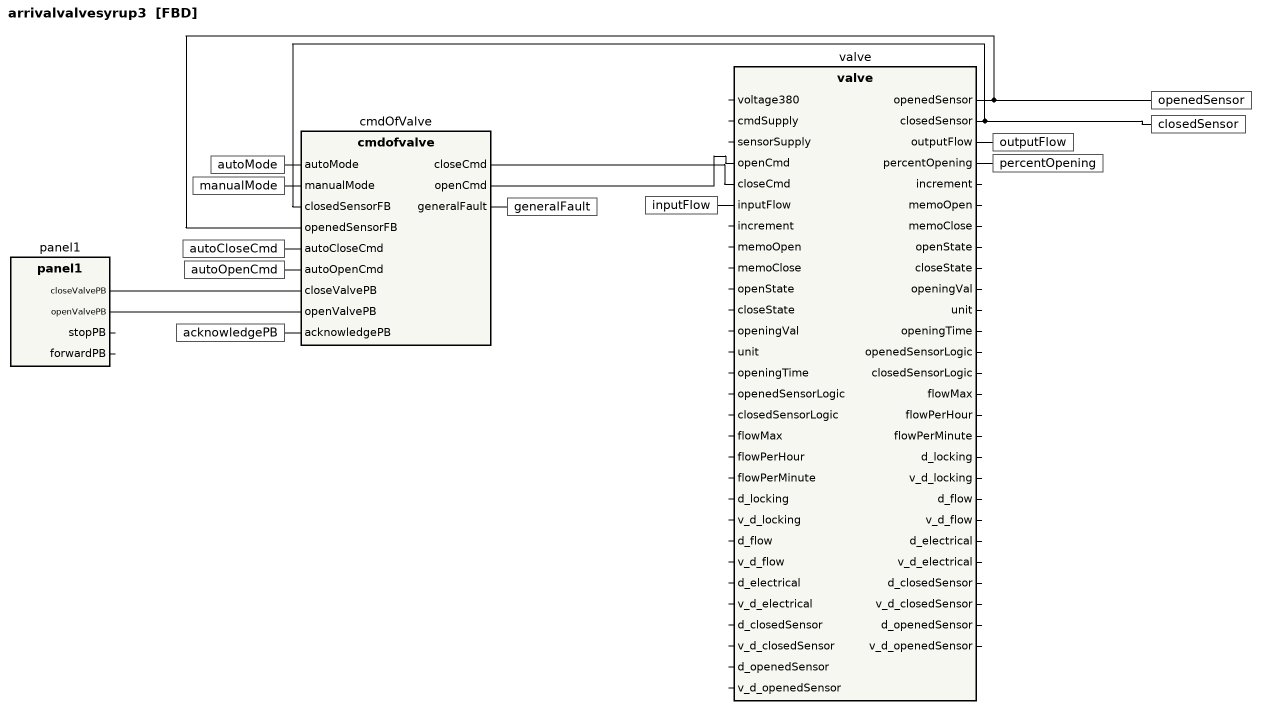
(* FBD diagram, written out as Structured Text *)
panel1();
cmdOfValve(autoMode := autoMode, manualMode := manualMode, closedSensorFB := valve.closedSensor, openedSensorFB := valve.openedSensor, autoCloseCmd := autoCloseCmd, autoOpenCmd := autoOpenCmd, closeValvePB := panel1.closeValvePB, openValvePB := panel1.openValvePB, acknowledgePB := acknowledgePB);
valve(openCmd := cmdOfValve.openCmd, closeCmd := cmdOfValve.closeCmd, inputFlow := inputFlow);
openedSensor := valve.openedSensor;
closedSensor := valve.closedSensor;
generalFault := cmdOfValve.generalFault;
outputFlow := valve.outputFlow;
percentOpening := valve.percentOpening;
END_PROGRAM

PROGRAM syrupextractionvalve
  VAR_INPUT
    acknowledgePB : BOOL := false;
    autoMode : BOOL := false;
    manualMode : BOOL := false;
    autoCloseCmd : BOOL := false;
    autoOpenCmd : BOOL := false;
    inputFlow : REAL := 0.0;
  END_VAR
  VAR_OUTPUT
    openedSensor : BOOL := false;
    closedSensor : BOOL := false;
    generalFault : BOOL := false;
    outputFlow : REAL := 0.0;
    percentOpening : REAL := 0.0;
  END_VAR

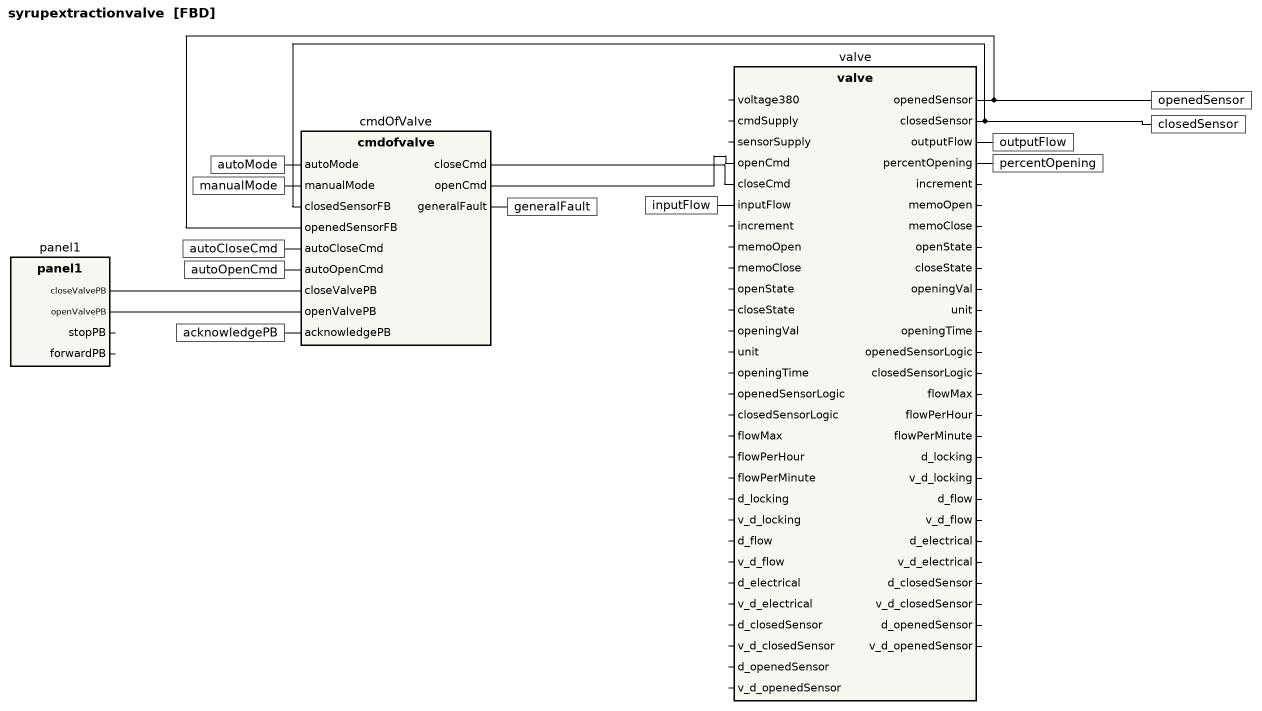
(* FBD diagram, written out as Structured Text *)
panel1();
cmdOfValve(autoMode := autoMode, manualMode := manualMode, closedSensorFB := valve.closedSensor, openedSensorFB := valve.openedSensor, autoCloseCmd := autoCloseCmd, autoOpenCmd := autoOpenCmd, closeValvePB := panel1.closeValvePB, openValvePB := panel1.openValvePB, acknowledgePB := acknowledgePB);
valve(openCmd := cmdOfValve.openCmd, closeCmd := cmdOfValve.closeCmd, inputFlow := inputFlow);
openedSensor := valve.openedSensor;
closedSensor := valve.closedSensor;
generalFault := cmdOfValve.generalFault;
outputFlow := valve.outputFlow;
percentOpening := valve.percentOpening;
END_PROGRAM

FUNCTION_BLOCK syrupmanagement
  VAR_INPUT
    weighingRequest : BOOL := false;
    cycleInProgress : BOOL := false;
    weighingWeight : INT := 0;
    syrup1Weight : INT := 0;
    syrup2Weight : INT := 0;
    syrup3Weight : INT := 0;
  END_VAR
  VAR_IN_OUT
    totalWeight : INT := 0;
    weighingS1 : BOOL := false;
    weighingS2 : BOOL := false;
    weighingS3 : BOOL := false;
    weighingS1Ok : BOOL := false;
    weighingS2Ok : BOOL := false;
    weighingS3Ok : BOOL := false;
    endOfWeighingS3 : BOOL := false;
    endOfWeighingS2 : BOOL := false;
    endOfWeighingS1 : BOOL := false;
    maxWeight : INT := 0;
  END_VAR
  VAR_OUTPUT
    weighingOk : BOOL := false;
    introduceS1 : BOOL := false;
    introS1End : BOOL := false;
    introduceS2 : BOOL := false;
    introS2End : BOOL := false;
    introduceS3 : BOOL := false;
    introS3End : BOOL := false;
    exitSyrup : BOOL := false;
    exitSyrupEnd : BOOL := false;
  END_VAR


ACTION C_source_code:

END_ACTION
END_FUNCTION_BLOCK

FUNCTION_BLOCK syrupquantity
  VAR_INPUT
    flowSyrup1 : REAL := 0.0;
    flowSyrup2 : REAL := 0.0;
    flowSyrup3 : REAL := 0.0;
  END_VAR
  VAR_OUTPUT
    flow : REAL := 0.0;
  END_VAR


ACTION C_source_code:

END_ACTION
END_FUNCTION_BLOCK

FUNCTION_BLOCK syrupstank
  VAR_INPUT
    inletFlow : REAL := 0.0;
    outletFlow : REAL := 0.0;
  END_VAR
  VAR_IN_OUT
    percent : REAL := 0.0;
    capacity : REAL := 0.0;
    d_level : BOOL := false;
    v_d_level : REAL := 0.0;
  END_VAR
  VAR_OUTPUT
    tankLevel : REAL := 0.0;
  END_VAR


ACTION C_source_code:

END_ACTION
END_FUNCTION_BLOCK

PROGRAM syrup
  VAR_INPUT
    syrup1Weight : INT := 0;
    syrup2Weight : INT := 0;
    syrup3Weight : INT := 0;
    cycleInProgress : BOOL := false;
    weighingRequest : BOOL := false;
    acknowledgePB : BOOL := false;
    autoMode : BOOL := false;
    manualMode : BOOL := false;
  END_VAR
  VAR_OUTPUT
    weighingOk : BOOL := false;
    fault : BOOL := false;
    syrupExtraction : REAL := 0.0;
  END_VAR

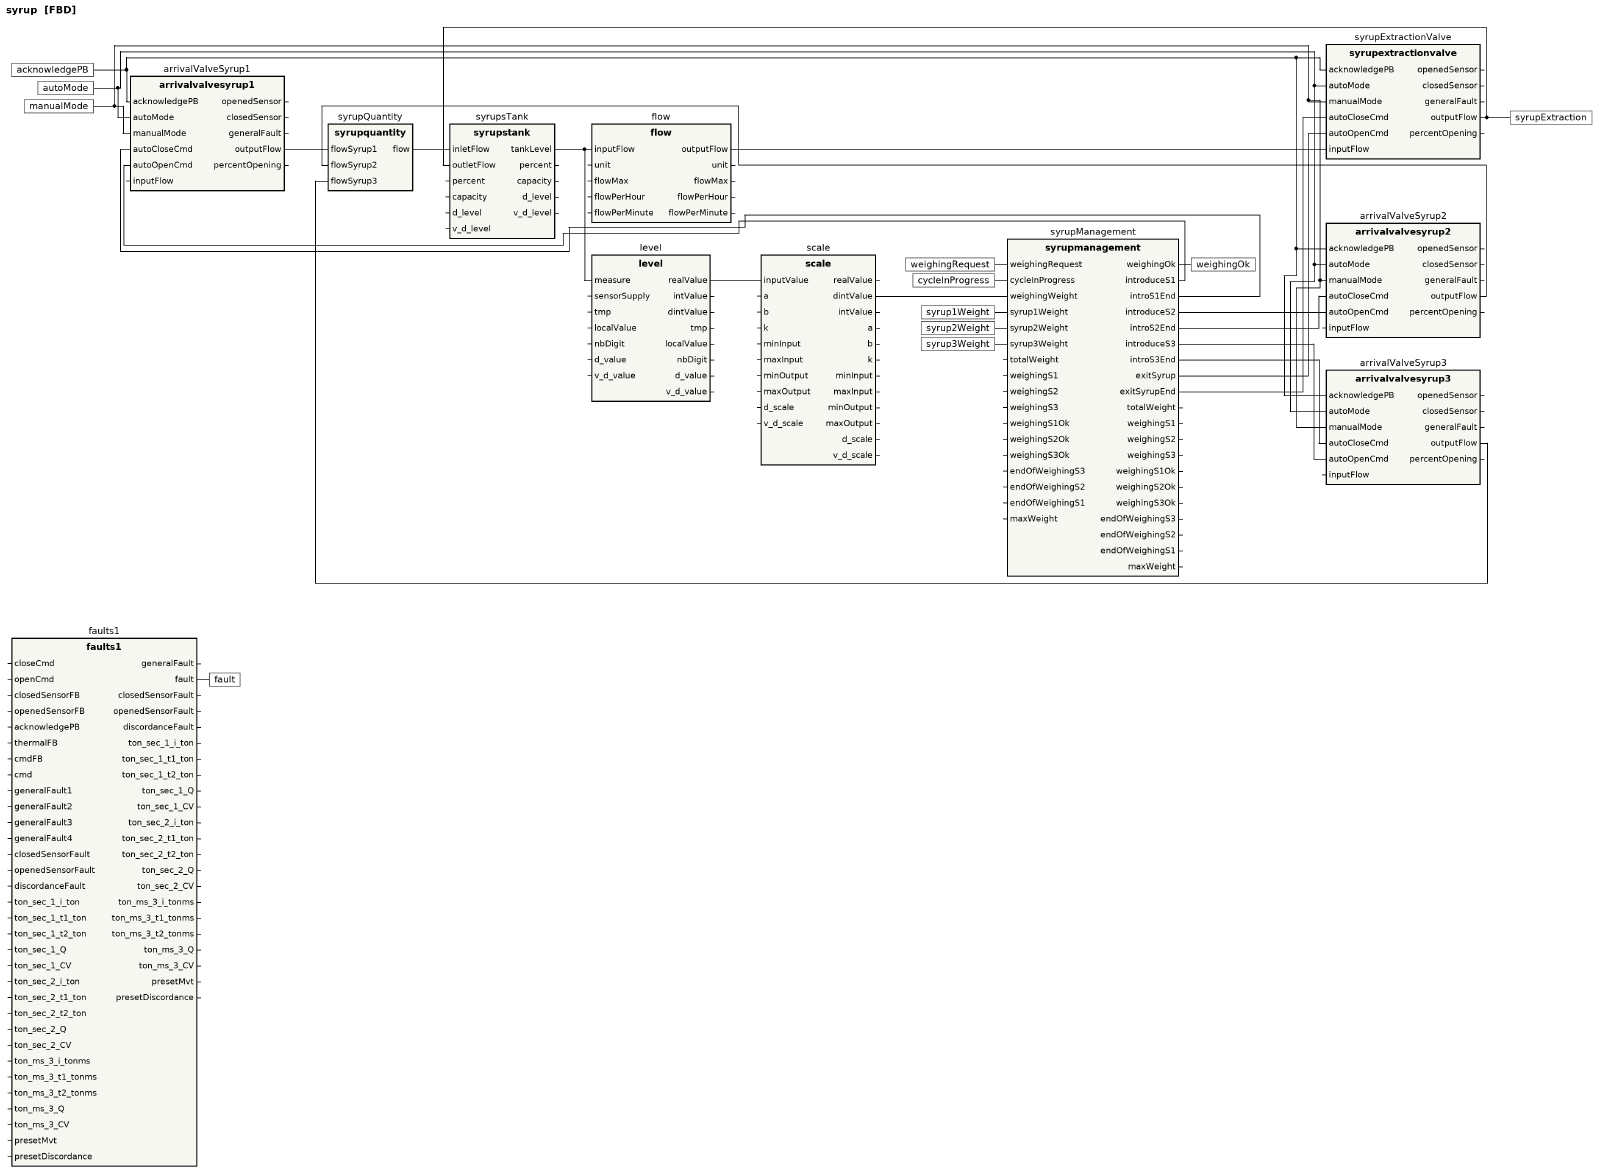
(* FBD diagram, written out as Structured Text *)
arrivalValveSyrup1(acknowledgePB := acknowledgePB, autoMode := autoMode, manualMode := manualMode, autoCloseCmd := syrupManagement.introS1End, autoOpenCmd := syrupManagement.introduceS1);
arrivalValveSyrup2(acknowledgePB := acknowledgePB, autoMode := autoMode, manualMode := manualMode, autoCloseCmd := syrupManagement.introS2End, autoOpenCmd := syrupManagement.introduceS2);
arrivalValveSyrup3(acknowledgePB := acknowledgePB, autoMode := autoMode, manualMode := manualMode, autoCloseCmd := syrupManagement.introS3End, autoOpenCmd := syrupManagement.introduceS3);
syrupQuantity(flowSyrup1 := arrivalValveSyrup1.outputFlow, flowSyrup2 := arrivalValveSyrup2.outputFlow, flowSyrup3 := arrivalValveSyrup3.outputFlow);
flow(inputFlow := syrupsTank.tankLevel);
syrupExtractionValve(acknowledgePB := acknowledgePB, autoMode := autoMode, manualMode := manualMode, autoCloseCmd := syrupManagement.exitSyrupEnd, autoOpenCmd := syrupManagement.exitSyrup, inputFlow := flow.outputFlow);
syrupsTank(inletFlow := syrupQuantity.flow, outletFlow := syrupExtractionValve.outputFlow);
level(measure := syrupsTank.tankLevel);
scale(inputValue := level.realValue);
syrupManagement(weighingRequest := weighingRequest, cycleInProgress := cycleInProgress, weighingWeight := scale.dintValue, syrup1Weight := syrup1Weight, syrup2Weight := syrup2Weight, syrup3Weight := syrup3Weight);
weighingOk := syrupManagement.weighingOk;
faults1();
fault := faults1.fault;
syrupExtraction := syrupExtractionValve.outputFlow;
END_PROGRAM

PROGRAM manufacturing
  VAR_INPUT
    cycleInProgress : BOOL := false;
    acknowledgePB : BOOL := false;
    flourWeighingRequest : BOOL := false;
    syrupWeighingRequest : BOOL := false;
    kneadingRequest : BOOL := false;
    autoMode : BOOL := false;
    manualMode : BOOL := false;
    flourWeight : INT := 0;
    syrup1Weight : INT := 0;
    syrup2Weight : INT := 0;
    syrup3Weight : INT := 0;
  END_VAR
  VAR_OUTPUT
    generalFault : BOOL := false;
    kneadingOK : BOOL := false;
    flourWeighingOk : BOOL := false;
    syrupWeighingOk : BOOL := false;
  END_VAR

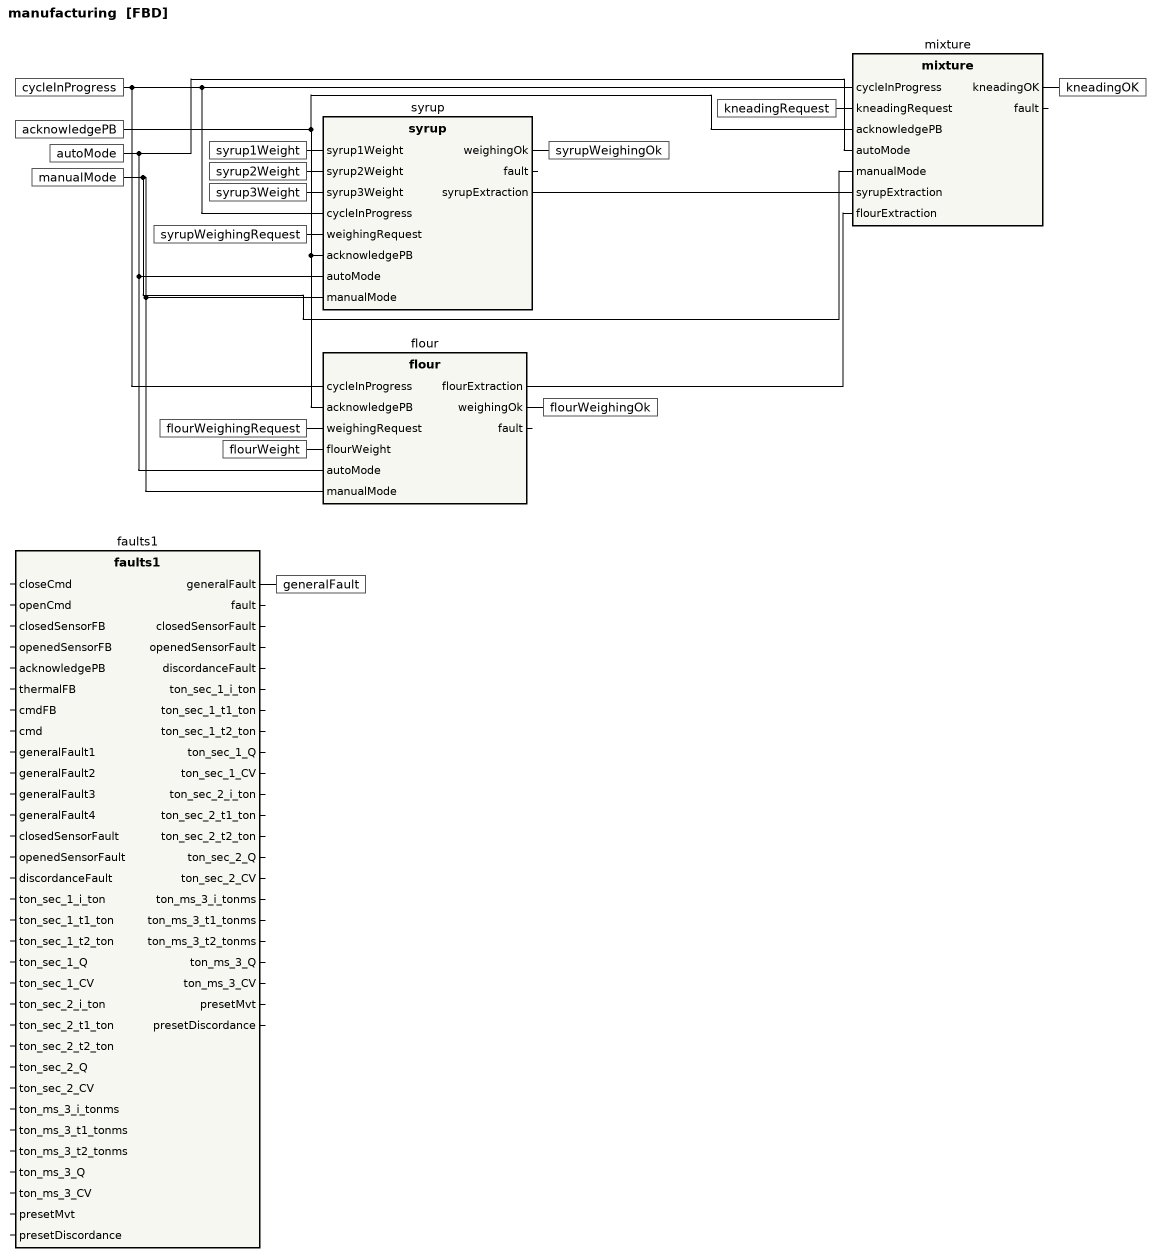
(* FBD diagram, written out as Structured Text *)
faults1();
generalFault := faults1.generalFault;
syrup(syrup1Weight := syrup1Weight, syrup2Weight := syrup2Weight, syrup3Weight := syrup3Weight, cycleInProgress := cycleInProgress, weighingRequest := syrupWeighingRequest, acknowledgePB := acknowledgePB, autoMode := autoMode, manualMode := manualMode);
flour(cycleInProgress := cycleInProgress, acknowledgePB := acknowledgePB, weighingRequest := flourWeighingRequest, flourWeight := flourWeight, autoMode := autoMode, manualMode := manualMode);
mixture(cycleInProgress := cycleInProgress, kneadingRequest := kneadingRequest, acknowledgePB := acknowledgePB, autoMode := autoMode, manualMode := manualMode, syrupExtraction := syrup.syrupExtraction, flourExtraction := flour.flourExtraction);
kneadingOK := mixture.kneadingOK;
flourWeighingOk := flour.weighingOk;
syrupWeighingOk := syrup.weighingOk;
END_PROGRAM

FUNCTION_BLOCK recipe
  VAR_IN_OUT
    recipeNumber : INT := 0;
  END_VAR
  VAR_OUTPUT
    flourWeight : INT := 0;
    syrup1Weight : INT := 0;
    syrup2Weight : INT := 0;
    syrup3Weight : INT := 0;
  END_VAR


ACTION C_source_code:

END_ACTION
END_FUNCTION_BLOCK

FUNCTION_BLOCK workingmodes
  VAR_INPUT
    powerUp : BOOL := false;
    emergencyStop : BOOL := false;
    manualSwitch : BOOL := false;
    autoSwitch : BOOL := false;
    startCyclePB : BOOL := false;
    endCyclePB : BOOL := false;
    acknowledgePB : BOOL := false;
    cycleEnd : BOOL := false;
    generalFault : BOOL := false;
  END_VAR
  VAR_IN_OUT
    emergencyStopState : BOOL := false;
  END_VAR
  VAR_OUTPUT
    live : BOOL := false;
    autoMode : BOOL := false;
    manualMode : BOOL := false;
    cycleInProgress : BOOL := false;
    endCycleRequest : BOOL := false;
  END_VAR


ACTION C_source_code:

END_ACTION
END_FUNCTION_BLOCK

PROGRAM my_app.batch

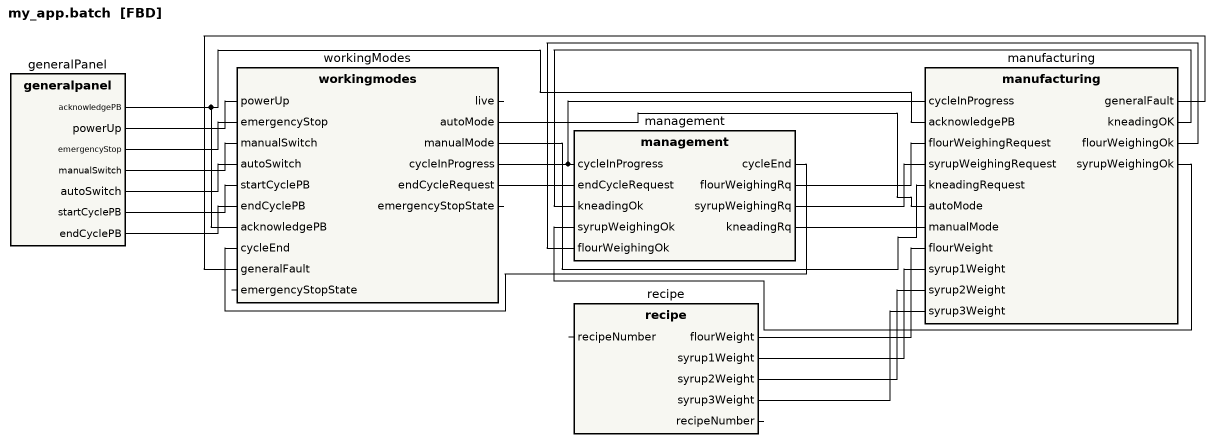
(* FBD diagram, written out as Structured Text *)
generalPanel();
management(cycleInProgress := workingModes.cycleInProgress, endCycleRequest := workingModes.endCycleRequest, kneadingOk := manufacturing.kneadingOK, syrupWeighingOk := manufacturing.syrupWeighingOk, flourWeighingOk := manufacturing.flourWeighingOk);
workingModes(powerUp := generalPanel.powerUp, emergencyStop := generalPanel.emergencyStop, manualSwitch := generalPanel.manualSwitch, autoSwitch := generalPanel.autoSwitch, startCyclePB := generalPanel.startCyclePB, endCyclePB := generalPanel.endCyclePB, acknowledgePB := generalPanel.acknowledgePB, cycleEnd := management.cycleEnd, generalFault := manufacturing.generalFault);
recipe();
manufacturing(cycleInProgress := workingModes.cycleInProgress, acknowledgePB := generalPanel.acknowledgePB, flourWeighingRequest := management.flourWeighingRq, syrupWeighingRequest := management.syrupWeighingRq, kneadingRequest := management.kneadingRq, autoMode := workingModes.autoMode, manualMode := workingModes.manualMode, flourWeight := recipe.flourWeight, syrup1Weight := recipe.syrup1Weight, syrup2Weight := recipe.syrup2Weight, syrup3Weight := recipe.syrup3Weight);
END_PROGRAM
